PROGRAM RunTests
VAR
    fbAtomicMassLookup_Test : FB_AtomicMassLookup_Test;
    fbAtomicNumberLookup_Test : FB_AtomicNumberLookup_Test;
    fbCalculateMassAttenuationCoefficient_Test : FB_CalculateXrayAbsorptionConstant_Test;
    fbCalculateThicknessFromTransmission_Test : FB_CalculateThicknessFromTransmission_Test;
    fbScatteringFactorLookupCXRO_Test : FB_ScatteringFactorLookupCXRO_Test;
    fbScatteringFactorLUT_Test : FB_ScatteringFactorLUT_Test;
    fbTestTransmission : FB_TestTransmission;
    fbTestElementDensity : FB_TestElementDensity;
    fbAtomicNumber_Test : FB_AtomicNumber_Test;

    (* Smoke test - just instantiate *)
    fbPhysicalConstants : FB_PhysicalConstants;
    fbAtomicMass : FB_AtomicMass;

END_VAR


TcUnit.RUN();

fbPhysicalConstants();
fbAtomicMass();

END_PROGRAM

(* stored: Version 1.1.0.1
   POU RunTests: Id {3c99bab2-48fb-4f3c-ae2b-1547c32b95ba}, SpecialFunc None *)
